(* PLC project Script Engine Example.project, CODESYS CODESYS V3.5 SP20 Patch 1 *)
(* stored: creationDateTime 2025-05-27T13:20:07.2176472, modificationDateTime 2025-05-06T14:40:48.6128089 *)

PROGRAM PLC_PRG

                    // Some boiler plate code
                  
END_PROGRAM

CONFIGURATION Device
  RESOURCE Application ON PLC
    TASK MainTask(INTERVAL := T#20ms, PRIORITY := 1);
    PROGRAM PLC_PRG WITH MainTask : PLC_PRG;
  END_RESOURCE
END_CONFIGURATION
